// TIA Portal project "FactoryIO_Template_S7-1200_V16_V16" (V16)
// Vorlageprojekt für das Buch mit Zielsystem S7-1200

(* hardware
DEVICE "S7-1200-Station_1"  S7-1200 Station
   slot 0: "Baugruppenträger_0"  Rack  V1.0
   slot 1: "PLC_1"  CPU 1211C DC/DC/DC  6ES7 211-1AE40-0XB0  V4.1
*)

// ===== PLC "PLC_1"  CPU 1211C DC/DC/DC =====

VAR_GLOBAL   // PLC tag table "Standard-Variablentabelle"
   "belt conveyor 2" AT %A0.0 : Bool;
   "start" AT %E0.0 : Bool;
   "stop" AT %E0.1 : Bool;
   "Tag_4" AT %I10.0 : Bool;
   "Tag_5" AT %Q10.0 : Bool;
   "Tag_6" AT %I10.1 : Bool;
   "elevator (right)" AT %I0.2 : Bool;
   "elevator (left)" AT %I0.3 : Bool;
   "inductive sensor 1" AT %I0.4 : Bool;
   "inductive sensor 2" AT %I0.5 : Bool;
   "belt conveyor 4" AT %Q0.1 : Bool;
   "belt conveyor  6" AT %Q0.2 : Bool;
   "elevator up" AT %Q0.3 : Bool;
   "elevator down" AT %Q0.4 : Bool;
   "elevator +" AT %Q0.5 : Bool;
   "start buttor light" AT %Q0.6 : Bool;
   "stop buttor light" AT %Q0.7 : Bool;
   "loop marker" AT %M0.0 : Bool;
   "Tag_1" AT %M0.1 : Bool;
   "Tag_2" AT %M0.2 : Bool;
   "Tag_3" AT %M0.3 : Bool;
   "Tag_7" AT %M0.4 : Bool;
   "Tag_8" AT %M0.5 : Bool;
END_VAR

FUNCTION "MHJ-PLC-Lab-Function-S71200" : Void   // FC9000, SCL
{ S7_Optimized_Access := 'TRUE' }
VERSION : 0.1
   VAR_TEMP
      rdTimeReturn : Int;
      outputTime : DTL;
      SyncVal : Byte;
      forVal : Int;
      forVal_2 : Int;
      Value : Byte;
   END_VAR
   VAR CONSTANT
      CompVal : Byte := 16#34;
      Value_01 : Byte := 16#11;
      Value_01_DW : DWord := 16#A165_D992;
      Value_02_DW : DWord := 16#58BE_4401;
   END_VAR
BEGIN

   #Value:=PEEK(area := 16#82,
        dbNumber := 0,
        byteOffset := 511);
   #Value := #Value + 1;

   POKE(area := 16#82,
        dbNumber := 0,
        byteOffset := 511,
        value := #Value);

   POKE(area:=16#81,
        dbNumber:=0,
        byteOffset:=1016,
        value:=#Value_01_DW);
   POKE(area := 16#81,
        dbNumber := 0,
        byteOffset := 1020,
        value := #Value_02_DW);

   POKE(area := 16#81,
        dbNumber := 0,
        byteOffset := 511,
        value := B#16#00);

   FOR #forVal := 0 TO 120 DO
       FOR #forVal_2:=0 TO 10 DO
           #rdTimeReturn:=RD_SYS_T(#outputTime);
           #rdTimeReturn := WR_SYS_T(#outputTime);
           #rdTimeReturn := RD_SYS_T(#outputTime);
           #rdTimeReturn := WR_SYS_T(#outputTime);
       END_FOR;
       #SyncVal:= PEEK(area := 16#81,
                      dbNumber := 0,
                      byteOffset := 511);
       IF #SyncVal = #CompVal THEN
          GOTO M_1;
       END_IF;
   END_FOR;
   RETURN;

   M_1:
   POKE(area := 16#81,
        dbNumber := 0,
        byteOffset := 511,
        value := B#16#0);
END_FUNCTION

ORGANIZATION_BLOCK "Main"   // OB1, LAD, ProgramCycle
TITLE = "Main Program Sweep (Cycle)"
{ S7_Optimized_Access := 'TRUE' }
VERSION : 0.1
   VAR_INPUT
      Initial_Call : Bool;   // Initial call of this OB
      Remanence : Bool;   // =True, if remanent data are available
   END_VAR
BEGIN

REGION Network 1: Konnektierungsbaustein für PLC-Lab
   // Im Netzwerk 1 wird der Konnektierungsbaustein für PLC-Lab aufgerufen.
   // Dieser Aufruf darf nicht entfernt werden!
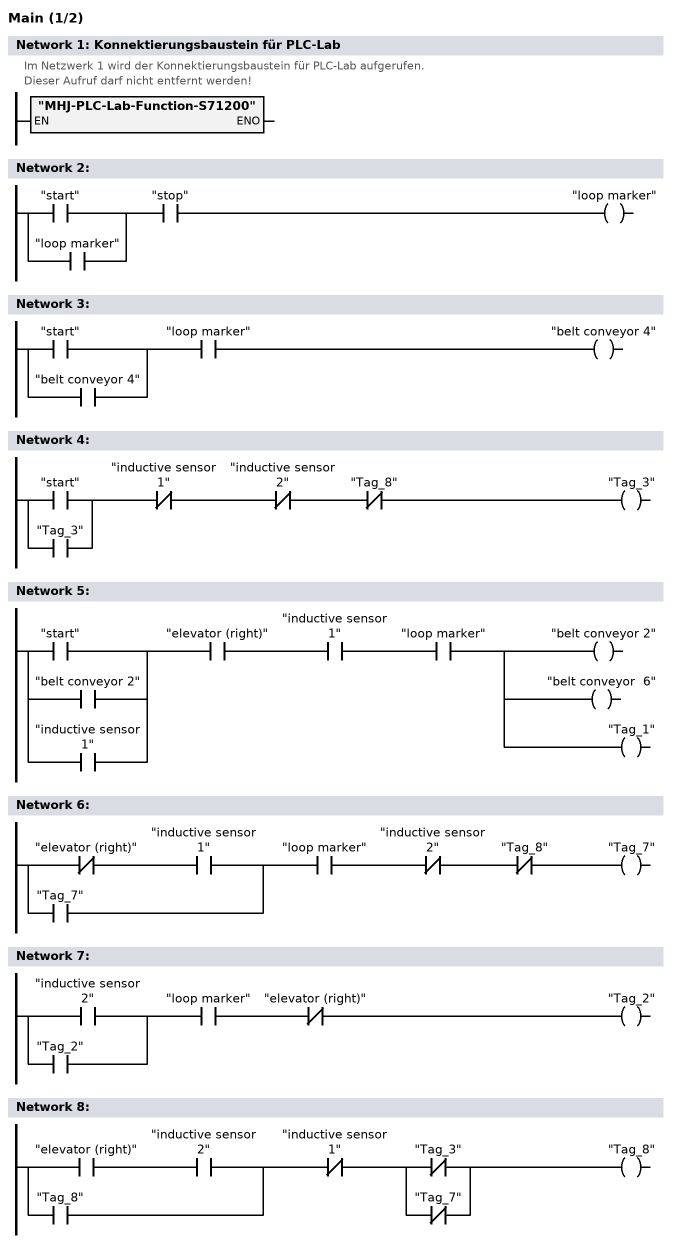
   RUNG wire#powerrail
      "MHJ-PLC-Lab-Function-S71200"()
   END_RUNG
   // the same network as SCL:
   "MHJ-PLC-Lab-Function-S71200"();
END_REGION

REGION Network 2
   RUNG wire#powerrail
      Contact( "start" )
      wire#w1
      Contact( "stop" )
      Coil( "loop marker" )
   END_RUNG
   RUNG wire#powerrail
      Contact( "loop marker" )
   END_RUNG wire#w1
   // the same network as SCL:
   "loop marker" := ("start" OR "loop marker") AND "stop";
END_REGION

REGION Network 3
   RUNG wire#powerrail
      Contact( "start" )
      wire#w1
      Contact( "loop marker" )
      Coil( "belt conveyor 4" )
   END_RUNG
   RUNG wire#powerrail
      Contact( "belt conveyor 4" )
   END_RUNG wire#w1
   // the same network as SCL:
   "belt conveyor 4" := ("start" OR "belt conveyor 4") AND "loop marker";
END_REGION

REGION Network 4
   RUNG wire#powerrail
      Contact( "start" )
      wire#w1
      I_Contact( "inductive sensor 1" )
      I_Contact( "inductive sensor 2" )
      I_Contact( "Tag_8" )
      Coil( "Tag_3" )
   END_RUNG
   RUNG wire#powerrail
      Contact( "Tag_3" )
   END_RUNG wire#w1
   // the same network as SCL:
   "Tag_3" := ("start" OR "Tag_3") AND NOT "inductive sensor 1" AND NOT "inductive sensor 2" AND NOT "Tag_8";
END_REGION

REGION Network 5
   RUNG wire#powerrail
      Contact( "start" )
      wire#w1
      Contact( "elevator (right)" )
      Contact( "inductive sensor 1" )
      Contact( "loop marker" )
      wire#w2
      Coil( "belt conveyor 2" )
   END_RUNG
   RUNG wire#powerrail
      Contact( "belt conveyor 2" )
   END_RUNG wire#w1
   RUNG wire#powerrail
      Contact( "inductive sensor 1" )
   END_RUNG wire#w1
   RUNG wire#w2
      Coil( "belt conveyor  6" )
   END_RUNG
   RUNG wire#w2
      Coil( "Tag_1" )
   END_RUNG
   // the same network as SCL:
   "belt conveyor 2" := ("start" OR "belt conveyor 2" OR "inductive sensor 1") AND "elevator (right)" AND "inductive sensor 1" AND "loop marker";
   "belt conveyor  6" := "belt conveyor 2";
   "Tag_1" := "belt conveyor 2";
END_REGION

REGION Network 6
   RUNG wire#powerrail
      I_Contact( "elevator (right)" )
      Contact( "inductive sensor 1" )
      wire#w1
      Contact( "loop marker" )
      I_Contact( "inductive sensor 2" )
      I_Contact( "Tag_8" )
      Coil( "Tag_7" )
   END_RUNG
   RUNG wire#powerrail
      Contact( "Tag_7" )
   END_RUNG wire#w1
   // the same network as SCL:
   "Tag_7" := ((NOT "elevator (right)" AND "inductive sensor 1") OR "Tag_7") AND "loop marker" AND NOT "inductive sensor 2" AND NOT "Tag_8";
END_REGION

REGION Network 7
   RUNG wire#powerrail
      Contact( "inductive sensor 2" )
      wire#w1
      Contact( "loop marker" )
      I_Contact( "elevator (right)" )
      Coil( "Tag_2" )
   END_RUNG
   RUNG wire#powerrail
      Contact( "Tag_2" )
   END_RUNG wire#w1
   // the same network as SCL:
   "Tag_2" := ("inductive sensor 2" OR "Tag_2") AND "loop marker" AND NOT "elevator (right)";
END_REGION

REGION Network 8
   RUNG wire#powerrail
      Contact( "elevator (right)" )
      Contact( "inductive sensor 2" )
      wire#w1
      I_Contact( "inductive sensor 1" )
      wire#w2
      I_Contact( "Tag_3" )
      wire#w3
      Coil( "Tag_8" )
   END_RUNG
   RUNG wire#powerrail
      Contact( "Tag_8" )
   END_RUNG wire#w1
   RUNG wire#w2
      I_Contact( "Tag_7" )
   END_RUNG wire#w3
   // the same network as SCL:
   "Tag_8" := (("elevator (right)" AND "inductive sensor 2") OR "Tag_8") AND NOT "inductive sensor 1" AND (NOT "Tag_3" OR NOT "Tag_7");
END_REGION

REGION Network 9
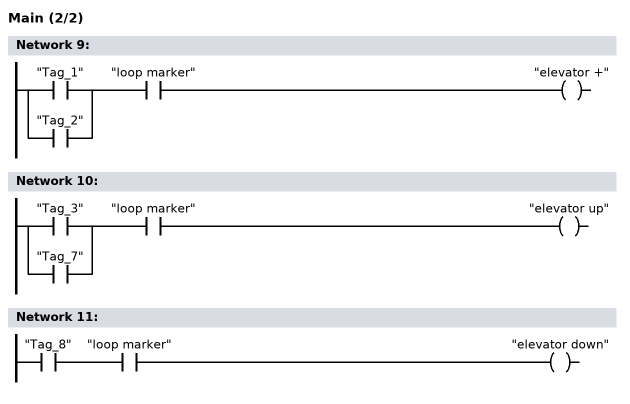
   RUNG wire#powerrail
      Contact( "Tag_1" )
      wire#w1
      Contact( "loop marker" )
      Coil( "elevator +" )
   END_RUNG
   RUNG wire#powerrail
      Contact( "Tag_2" )
   END_RUNG wire#w1
   // the same network as SCL:
   "elevator +" := ("Tag_1" OR "Tag_2") AND "loop marker";
END_REGION

REGION Network 10
   RUNG wire#powerrail
      Contact( "Tag_3" )
      wire#w1
      Contact( "loop marker" )
      Coil( "elevator up" )
   END_RUNG
   RUNG wire#powerrail
      Contact( "Tag_7" )
   END_RUNG wire#w1
   // the same network as SCL:
   "elevator up" := ("Tag_3" OR "Tag_7") AND "loop marker";
END_REGION

REGION Network 11
   RUNG wire#powerrail
      Contact( "Tag_8" )
      Contact( "loop marker" )
      Coil( "elevator down" )
   END_RUNG
   // the same network as SCL:
   "elevator down" := "Tag_8" AND "loop marker";
END_REGION
END_ORGANIZATION_BLOCK